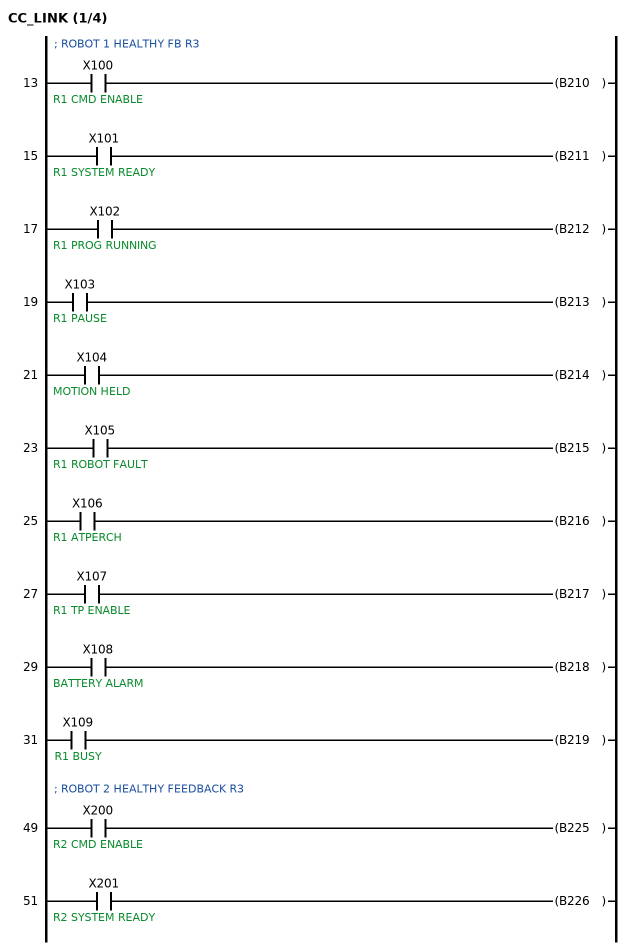
[picture p24: ladder of CC_LINK, rungs at steps 13 to 51]
; ROBOT 1 HEALTHY FB R3
13    LD      X100  ; R1 CMD ENABLE
      OUT     B210
15    LD      X101  ; R1 SYSTEM READY
      OUT     B211
17    LD      X102  ; R1 PROG RUNNING
      OUT     B212
19    LD      X103  ; R1 PAUSE
      OUT     B213
21    LD      X104  ; MOTION HELD
      OUT     B214
23    LD      X105  ; R1 ROBOT FAULT
      OUT     B215
25    LD      X106  ; R1 ATPERCH
      OUT     B216
27    LD      X107  ; R1 TP ENABLE
      OUT     B217
29    LD      X108  ; BATTERY ALARM
      OUT     B218
31    LD      X109  ; R1 BUSY
      OUT     B219
; ROBOT 2 HEALTHY FEEDBACK R3
49    LD      X200  ; R2 CMD ENABLE
      OUT     B225
51    LD      X201  ; R2 SYSTEM READY
      OUT     B226
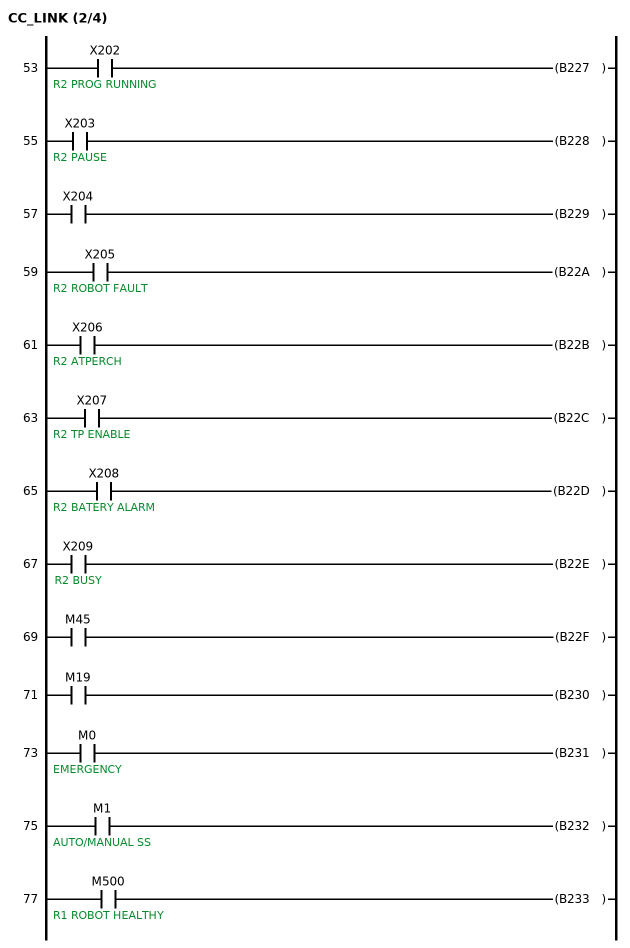
53    LD      X202  ; R2 PROG RUNNING
      OUT     B227
55    LD      X203  ; R2 PAUSE
      OUT     B228
57    LD      X204
      OUT     B229
59    LD      X205  ; R2 ROBOT FAULT
      OUT     B22A
61    LD      X206  ; R2 ATPERCH
      OUT     B22B
63    LD      X207  ; R2 TP ENABLE
      OUT     B22C
65    LD      X208  ; R2 BATERY ALARM
      OUT     B22D
67    LD      X209  ; R2 BUSY
      OUT     B22E
69    LD      M45
      OUT     B22F
71    LD      M19
      OUT     B230
73    LD      M0  ; EMERGENCY
      OUT     B231
75    LD      M1  ; AUTO/MANUAL SS
      OUT     B232
77    LD      M500  ; R1 ROBOT HEALTHY
      OUT     B233
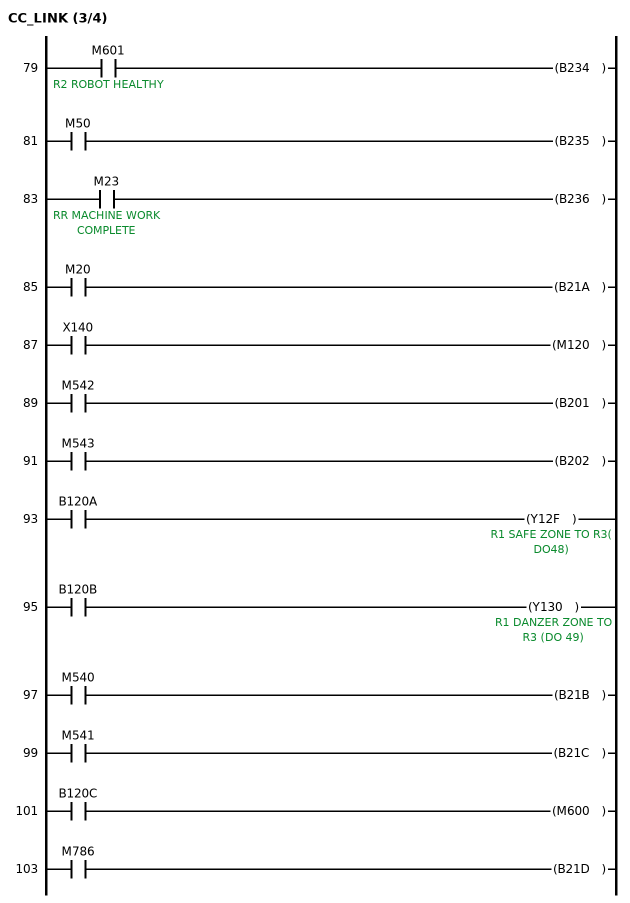
79    LD      M601  ; R2 ROBOT HEALTHY
      OUT     B234
81    LD      M50
      OUT     B235
83    LD      M23  ; RR MACHINE WORK COMPLETE
      OUT     B236
85    LD      M20
      OUT     B21A
87    LD      X140
      OUT     M120
89    LD      M542
      OUT     B201
91    LD      M543
      OUT     B202
93    LD      B120A
      OUT     Y12F  ; R1 SAFE ZONE TO R3( DO48)
95    LD      B120B
      OUT     Y130  ; R1 DANZER ZONE TO R3 (DO 49)
97    LD      M540
      OUT     B21B
99    LD      M541
      OUT     B21C
101   LD      B120C
      OUT     M600
103   LD      M786
      OUT     B21D
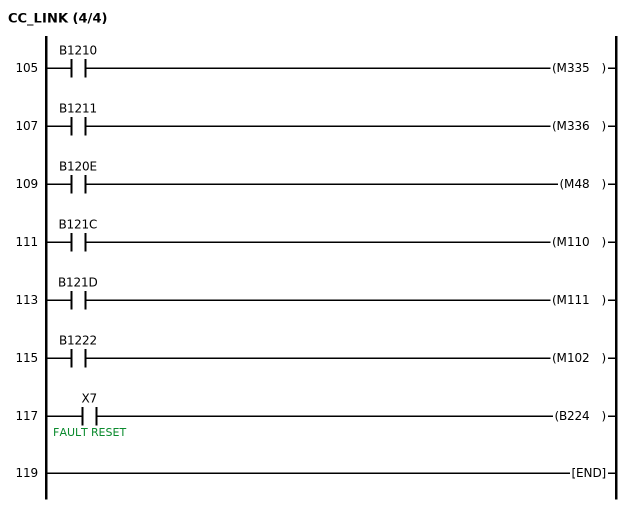
105   LD      B1210
      OUT     M335
107   LD      B1211
      OUT     M336
109   LD      B120E
      OUT     M48
111   LD      B121C
      OUT     M110
113   LD      B121D
      OUT     M111
115   LD      B1222
      OUT     M102
117   LD      X7  ; FAULT RESET
      OUT     B224
119   END
END_PROGRAM

PROGRAM ZONNING
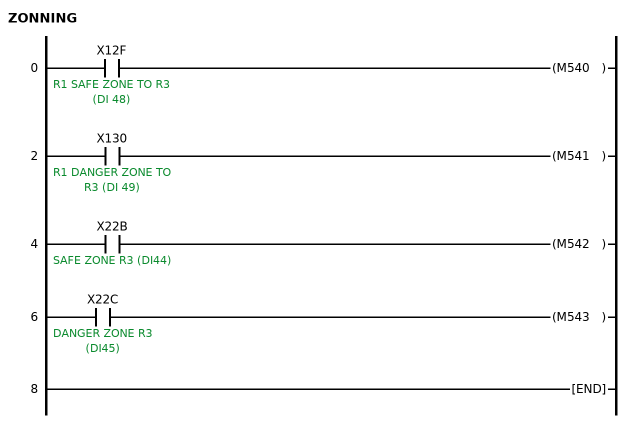
0     LD      X12F  ; R1 SAFE ZONE TO R3 (DI 48)
      OUT     M540
2     LD      X130  ; R1 DANGER ZONE TO R3 (DI 49)
      OUT     M541
4     LD      X22B  ; SAFE ZONE R3 (DI44)
      OUT     M542
6     LD      X22C  ; DANGER ZONE R3 (DI45)
      OUT     M543
8     END
END_PROGRAM

// device comments not shown above
X10A  ; R1 RSR 1 HIGH TEM
X10B  ; R1 RSR 2 LOW TEM
X10C  ; R1 RSR 1 OK TEM
X131  ; GREEPER OPEN CMD
X150  ; ROBOT 2 SAFE ZONE
X22D  ; SAFE ZONE TO R2
X22E  ; DANZER ZONE TO R2
X23D  ; WORK COMPLETE TO RR      (DI62)
Y203  ; R2 CYCLE STOP
Y209  ; RSR 2
Y22D  ; SAFE ZONE 2 R2
Y22E  ; DANZER ZONE TO R2
Y232  ; ROBOT 2 SAFE ZONE
Y233  ; ROBOT 3 DANGER ZONE
Y234  ; ROBOT 2 WORK COMPLETE
Y400  ; R3 IMSTP
Y401  ; R3 HOLD
Y402  ; R3 SFS
Y403  ; R3 CYCLE STOP
Y404  ; R3 FAULT RESET
Y405  ; R3 START
Y407  ; R3 ENABLE
Y408  ; RSR 1
Y409  ; RSR 2
M510  ; COIL MBIT 1
M700  ; R3 ROBOT HEALTHY
